TYPE ST_MasterData :
STRUCT
	ID						: WORD;
	Name					: STRING;
	Status					: STRING;
	NetId					: T_AmsNetId;
	LostFrames     			: UDINT;
	FramesPerSecond        	: LREAL;
	LostQueuedFrames      	: UDINT;
	QueuedFramesPerSecond 	: LREAL;
END_STRUCT
END_TYPE

(* stored: Version 1.1.0.1, ProductVersion 3.1.4024.3
   DUT ST_MasterData: Id {0fe86ee6-b7f5-466e-9869-07da82261196} *)
